FUNCTION_BLOCK strip_set_pixel (* Service Interface Function Block Type *)
  (* Standard: 61499-2 *)
  (* Version 1.0, 2022-07-16, franz *)
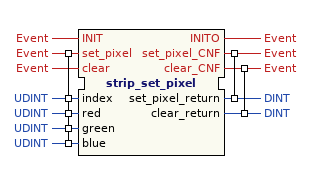
  EVENT_INPUT
    INIT; (* Service Initialization *)
    set_pixel WITH index, red, green, blue; (* Set RGB for a specific pixel *)
    clear; (* Clear LED strip (turn off all LEDs) *)
  END_EVENT
  EVENT_OUTPUT
    INITO; (* Initialization Confirm *)
    set_pixel_CNF WITH set_pixel_return; (* Confirmation of set_pixel *)
    clear_CNF WITH clear_return; (* Confirmation of clear *)
  END_EVENT
  VAR_INPUT
    index : UDINT; (* index of pixel to set *)
    red : UDINT; (* red part of color *)
    green : UDINT; (* green part of color *)
    blue : UDINT; (* blue part of color *)
  END_VAR
  VAR_OUTPUT
    set_pixel_return : DINT; (* Error indication *)
    clear_return : DINT;
  END_VAR
  SERVICE APPLICATION/RESOURCE (* Service Interface Function Block Type *)
    SEQUENCE normal_establishment
      APPLICATION.INIT+(PARAMS) -> RESOURCE.initialize(PARAMS) -> APPLICATION.INITO+();
    END_SEQUENCE
    SEQUENCE unsuccessful_establishment
      APPLICATION.INIT+(PARAMS) -> RESOURCE.initialize(PARAMS) -> APPLICATION.INITO-(STATUS);
    END_SEQUENCE
    SEQUENCE request_confirm
      APPLICATION.REQ+(SD) -> RESOURCE.request(SD) -> APPLICATION.CNF+(RD);
    END_SEQUENCE
    SEQUENCE request_inhibited
      APPLICATION.REQ-(SD) -> APPLICATION.CNF-(STATUS);
    END_SEQUENCE
    SEQUENCE request_error
      APPLICATION.REQ+(SD) -> RESOURCE.request(SD) -> APPLICATION.CNF-(STATUS);
    END_SEQUENCE
    SEQUENCE indication_response
      RESOURCE.indicate(RD) -> APPLICATION.IND+(RD);
      APPLICATION.RSP(QI,SD) -> RESOURCE.response(QI,SD);
    END_SEQUENCE
    SEQUENCE indication_inhibited
      RESOURCE.indicate(RD,QI=FALSE) -> RESOURCE.inhibited();
    END_SEQUENCE
    SEQUENCE error_indication
      RESOURCE.error(STATUS) -> APPLICATION.IND-(STATUS);
    END_SEQUENCE
    SEQUENCE application_initiated_termination
      APPLICATION.INIT-() -> RESOURCE.terminate() -> APPLICATION.INITO-(STATUS);
    END_SEQUENCE
    SEQUENCE resource_initiated_termination
      -> APPLICATION.INITO-(STATUS);
    END_SEQUENCE
  END_SERVICE
END_FUNCTION_BLOCK
